FUNCTION_BLOCK ABSTRACT FB_AbstructContainerDynamicJob IMPLEMENTS I_Future, I_Container
VAR_INPUT
END_VAR
VAR_OUTPUT
END_VAR
VAR
	_executor : I_Job;
	{attribute 'TcEncoding':='UTF-8'}
	_name 	: STRING := 'BATCH JOB';
	_executors : ARRAY [1..ParamFuturesLib.MAX_TASK_NUM] OF I_Job;
	_start :BOOL;
	_auto_start : BOOL := TRUE;
	_abort : BOOL;
	_num_of_jobs: UDINT;
	_continuous_mode : BOOL;
	_error_id :HRESULT;
	_state :E_FutureExecutionState;
	_job_event_reporter : I_JobInfo;
END_VAR

METHOD PROTECTED _append_job : BOOL
VAR_INPUT
	executor	: I_Job;
END_VAR
END_METHOD

(* This is the generator that iteratively generates references to FB_executor instances*)
METHOD _index_generator_ : UINT
VAR_INST
	_index : UINT;
END_VAR
_index := _index + 1;
IF _index > _num_of_jobs THEN
	_index := 0;
END_IF
_index_generator_ := _index;
END_METHOD

METHOD abort : BOOL // Return TRUE if finish.
END_METHOD

METHOD append_job : BOOL
VAR_INPUT
	executor	: I_Job;
END_VAR
executor.persistent_job := TRUE;
THIS^._append_job(executor);
END_METHOD

{warning 'Add property implementation'}
PROPERTY auto_start : BOOL
GET
auto_start := _auto_start;
END_GET
SET
_auto_start := auto_start;
END_SET
END_PROPERTY

PROPERTY continuous_mode : BOOL
SET
VAR
	_executor : I_Job;
END_VAR
_continuous_mode := continuous_mode;
REPEAT
	_executor := THIS^.each_executor;
	IF _executor <> 0 THEN
		_executor.continuous_mode := continuous_mode;
	END_IF
UNTIL
	_executor = 0
END_REPEAT
END_SET
END_PROPERTY

METHOD create_container : I_Job
VAR_INPUT
	container_type	: ContainerType;
	name	: STRING;
END_VAR
CASE container_type OF
	ContainerType.BATCH:
		create_container := THIS^.create_job(GVL.batch_job_container_creator,name);
	ContainerType.PARALLEL:
		create_container := THIS^.create_job(GVL.parallel_job_container_creator,name);
	ContainerType.QUEUE:
		create_container := THIS^.create_job(GVL.queue_job_container_creator,name);
	ContainerType.PARALLEL_QUEUE:
		create_container := THIS^.create_job(GVL.parallel_queue_job_container_creator,name);
END_CASE
END_METHOD

METHOD create_job : I_Job
VAR_INPUT
	creator	: I_TaskCreator;
	future_name	: STRING;
END_VAR
VAR
	future : I_Future;
END_VAR
IF _num_of_jobs < ParamFuturesLib.MAX_TASK_NUM THEN
	future := creator.create_future(future_name);
	create_job := THIS^.spawn_job(future);
	IF create_job <> 0 THEN
		create_job.future_creator := creator;
	ELSE
		creator.destroy_future(future);
	END_IF
END_IF
END_METHOD

PROPERTY each_executor : I_Job
GET
VAR
	_index : UINT;
END_VAR
_index := _index_generator_();
IF _index > 0 THEN
	IF _executors[_index] <> 0 THEN
		IF _executors[_index] <> 0 THEN
			each_executor := _executors[_index];
		ELSE
			each_executor := 0;
		END_IF
	END_IF
ELSE
	each_executor := 0;
END_IF
END_GET
END_PROPERTY

METHOD error_reset : BOOL
VAR
	_executor : I_Job;
	complete : BOOL;
END_VAR
complete := TRUE;
REPEAT
	_executor := each_executor;
	IF _executor <> 0 THEN
		IF NOT _executor.error_reset() THEN
			complete := FALSE;
		END_IF
	END_IF
UNTIL
	_executor = 0
END_REPEAT
IF complete THEN
	_error_id := 0;
END_IF
error_reset := complete;
END_METHOD

METHOD execute : BOOL // Return TRUE if finish.
END_METHOD

PROPERTY executor : I_Job
GET
executor := _executor;
END_GET
SET
_executor := executor;
END_SET
END_PROPERTY

PROPERTY future_name : STRING// Name of future.
GET
future_name := _name;
END_GET
SET
_name := future_name;
END_SET
END_PROPERTY

METHOD init : BOOL // Return TRUE if finish.
VAR
	_each_executor : i_Job;
	_init_done : BOOL;
END_VAR
_init_done := TRUE;
REPEAT
	_each_executor := THIS^.each_executor;
	IF _each_executor <> 0 THEN
		IF NOT _each_executor.init() THEN
			_init_done := FALSE;
		END_IF
	END_IF
UNTIL
	_each_executor = 0
END_REPEAT

_error_id := 0;
init := _init_done;
END_METHOD

PROPERTY nErrorID : HRESULT
GET
nErrorID := _error_id;
END_GET
END_PROPERTY

PROPERTY num_of_jobs : UDINT
GET
num_of_jobs := _num_of_jobs;
END_GET
END_PROPERTY

METHOD quit : BOOL // Return TRUE if finish.
quit := TRUE;
END_METHOD

METHOD reset : BOOL // Return TRUE if finish.
VAR_INPUT
	deep : BOOL := FALSE;
END_VAR
VAR
	i : UINT;
	_delete_counter : UINT;
	_p_executor : POINTER TO FB_Executor;
	text : STRING;
END_VAR
_delete_counter := 0;
REPEAT
	i := _index_generator_();
	IF _num_of_jobs > _delete_counter AND i > 0 THEN
		IF _executors[i] <> 0 THEN
			IF _executors[i].reset(deep) THEN
				IF _executors[i].persistent_job THEN
					_executors[i] := 0;
				ELSIF __QUERYPOINTER(_executors[i],_p_executor) THEN
					__DELETE(_p_executor);
				END_IF
				_delete_counter := _delete_counter + 1;
			END_IF
		END_IF
	END_IF
UNTIL
	i = 0
END_REPEAT
_num_of_jobs := _num_of_jobs - _delete_counter;
reset := _num_of_jobs = 0;
END_METHOD

METHOD resume : BOOL
VAR
	_all_done : BOOL;
END_VAR
VAR_INST
	_executor : I_Job;
END_VAR
_all_done := TRUE;
REPEAT
	_executor := THIS^.each_executor;
	IF _executor <> 0 THEN
		IF NOT _executor.resume() THEN
			_all_done := FALSE;
		END_IF
	END_IF
UNTIL
	_executor = 0
END_REPEAT
resume := _all_done;
END_METHOD

METHOD spawn_job : I_Job
VAR_INPUT
	future : I_Future;
END_VAR
VAR
	_spawned_executor : POINTER TO FB_Executor;
END_VAR
IF future <> 0 THEN
	_spawned_executor := __NEW(FB_Executor);
	_spawned_executor^.future := future;
	_spawned_executor^.persistent_job := FALSE;
	_append_job(_spawned_executor^);
	spawn_job := _spawned_executor^;
ELSE
	spawn_job := 0;
END_IF
END_METHOD

PROPERTY state : E_FutureExecutionState
GET
state := _state;
END_GET
SET
_state := state;
END_SET
END_PROPERTY

END_FUNCTION_BLOCK

(* stored: Version 1.1.0.1, ProductVersion 3.1.4026.17
   POU FB_AbstructContainerDynamicJob: Id {b670b0ef-80fd-4471-bcf6-273d9d0112e2}, SpecialFunc None
   Method _append_job: Id {d4d7e6e3-b98b-4b63-9ff1-5d7eecbfe649}
   Method _index_generator_: Id {db255ff0-959a-4e60-aa5a-e2c61cb1e8de}
   Method abort: Id {f45b039d-c15f-4eae-8016-a9f5a458d8d3}
   Method append_job: Id {cb2a0d16-d4ad-452d-8f0f-aa58703f0d60}
   Property auto_start: Id {a4d668e2-2876-4149-82f4-6184faf6aa75}
   Get Get: Id {8a55e905-c1ad-4870-a63a-fbd6945dc10b}
   Set Set: Id {7678fa7d-ae92-4fc5-bc1d-66bf25141c88}
   Property continuous_mode: Id {3c2e5149-af3c-4d7a-a5d6-b5f93fde7ff0}
   Set Set: Id {15e7a70f-2a85-4994-83b2-d2334b8070fc}
   Method create_container: Id {dfd7dce2-6d2c-4ad3-b58b-28fc111968f3}
   Method create_job: Id {6e2d3e38-0c5d-46f5-b4f8-ee01bcd4f24d}
   Property each_executor: Id {3dcd0647-7122-40e7-96be-29746514bf0d}
   Get Get: Id {1b542c98-0d01-48d6-bb16-6a442ffc0e43}
   Method error_reset: Id {103e8728-adc1-4801-ac51-6d8bf2e3e385}
   Method execute: Id {e6ad1c69-a35c-402b-b841-0ed974c585de}
   Property executor: Id {3b8baf7d-561a-4d10-8efb-1ae3d62c407a}
   Get Get: Id {738c4369-32ff-4055-b220-d86316d09cb8}
   Set Set: Id {efb40c42-376b-4ea8-aed4-6fe4a1d53cef}
   Property future_name: Id {5f975bd9-62df-4754-bbc5-1459be061c94}
   Get Get: Id {b4751c18-e95f-4c58-b987-0c5e90fe80e3}
   Set Set: Id {66b13ece-63e1-449e-aaff-d26bdd78023d}
   Method init: Id {12b7c49c-e051-46ee-b3a8-dbe1f20bf366}
   Property nErrorID: Id {d16d58c9-b0d2-4458-8e73-64e35e480136}
   Get Get: Id {13532608-6057-4343-9e7a-e7fddd1ab8ef}
   Property num_of_jobs: Id {29f71da5-b307-4261-85b8-e456a260849a}
   Get Get: Id {d733b605-14a6-450b-96a0-439bb558ddef}
   Method quit: Id {01690ddf-2fd1-42a0-b9cb-c5e873bd91b2}
   Method reset: Id {72ea1b7b-30d6-40f9-87bd-bc754c843ab3}
   Method resume: Id {cc30cf46-7981-43e6-8b94-9b85af441cf3}
   Method spawn_job: Id {638bf563-4ad7-49bb-b39c-ac9d7646466f}
   Property state: Id {7e6bca75-e6e9-43a5-96e4-74eefdde8672}
   Get Get: Id {9bca2c78-9788-4055-8249-802a71c99c79}
   Set Set: Id {98b60d06-5786-47e1-879d-b914f0519e29} *)
